FUNCTION_BLOCK FB_SimCapper EXTENDS FB_SimStation
VAR_INPUT
END_VAR
VAR_OUTPUT
END_VAR
VAR
	tmrWork						: TON;
END_VAR

METHOD PROTECTED  DoWork : BOOL
VAR_INPUT
END_VAR
tmrWork(IN:=TRUE, PT:=T#2S);
IF tmrWork.Q THEN
	tmrWork(IN:=FALSE);
	DoWork := TRUE;
END_IF
END_METHOD

METHOD PROTECTED  UpdatePartStatus : PVOID
VAR_INPUT
END_VAR
IF pPartStatus <> 0 THEN
	pPartStatus^.bCapperStatus := TRUE;
END_IF
END_METHOD

END_FUNCTION_BLOCK

(* stored: Version 1.1.0.1, ProductVersion 3.1.4024.12
   POU FB_SimCapper: Id {84003403-a58a-475b-b316-c108bd8518cd}, SpecialFunc None
   Method DoWork: Id {98a2339c-2826-4eac-a5b9-47f72a58485a}
   Method UpdatePartStatus: Id {69b5a33a-351a-4da4-957b-7d2171099c68} *)
